{attribute 'linkalways'} 
{attribute 'no_explicit_call' := 'This FB is a CLASS and must be accessed using methods or properties'}
{attribute 'enable_dynamic_creation'}
FUNCTION_BLOCK DatatypeOperations
VAR
	operations : Stack;
END_VAR

METHOD PUBLIC AddMemoryCopyOperation
VAR_INPUT
	Source : I_Datatype;
	Destination : I_Datatype;
END_VAR
VAR
	operation : I_DatatypeOperation;
END_VAR
operation := CreateMemoryCopyOperation(Source,Destination);
operations.Push(operation);
END_METHOD

METHOD PUBLIC AddSafeMemoryCopyOperation
VAR_INPUT
	Source : I_Datatype;
	Destination : I_Datatype;
END_VAR
VAR
	operation : I_DatatypeOperation;
END_VAR
operation := CreateSafeMemoryCopyOperation(Source,Destination);
operations.Push(operation);
END_METHOD

METHOD PUBLIC AddWriteBitToBoolOperation
VAR_INPUT
	Source : I_BitDatatype;
	Destination : Reference to _BOOL;
END_VAR
VAR
	operation : I_DatatypeOperation;
END_VAR
operation := CreateWriteBitToBoolOperation(Source,Destination);
operations.Push(operation);
END_METHOD

METHOD PUBLIC AddWriteBoolToBitOperation
VAR_INPUT
	Source : REFERENCE TO _BOOL;
	Destination : I_BitDatatype;
END_VAR
VAR
	operation : I_DatatypeOperation;
END_VAR
operation := CreateWriteBoolToBitOperation(Source,Destination);
operations.Push(operation);
END_METHOD

METHOD PUBLIC Clear
VAR
	operation : I_DatatypeOperation;
END_VAR
WHILE operations.TryPop(operation) DO
	operation.Dispose();
END_WHILE
END_METHOD

METHOD PRIVATE CreateMemoryCopyOperation : I_DatatypeOperation
VAR_INPUT
	OperationSource : I_Datatype;
	OperationDestination : I_Datatype;
END_VAR
VAR
	pOperation : POINTER TO MemCopyOperation;
END_VAR
pOperation := __NEW(MemCopyOperation(Source := OperationSource, Destination := OperationDestination));
CreateMemoryCopyOperation := pOperation^;
END_METHOD

METHOD PRIVATE CreateSafeMemoryCopyOperation : I_DatatypeOperation
VAR_INPUT
	OperationSource : I_Datatype;
	OperationDestination : I_Datatype;
END_VAR
VAR
	pOperation : POINTER TO SafeMemCopyOperation;
END_VAR
pOperation := __NEW(SafeMemCopyOperation(Source := OperationSource, Destination := OperationDestination));
CreateSafeMemoryCopyOperation := pOperation^;
END_METHOD

METHOD PRIVATE CreateWriteBitToBoolOperation : I_DatatypeOperation
VAR_INPUT
	OperationSource : I_BitDatatype;
	OperationDestination : REFERENCE TO _BOOL;
END_VAR
VAR
	pOperation : POINTER TO WriteBitToBoolOperation;
END_VAR
pOperation := __NEW(WriteBitToBoolOperation(Source := OperationSource, Destination := OperationDestination));
CreateWriteBitToBoolOperation := pOperation^;
END_METHOD

METHOD PRIVATE CreateWriteBoolToBitOperation : I_DatatypeOperation
VAR_INPUT
	OperationSource : REFERENCE TO _BOOL;
	OperationDestination : I_BitDatatype;
END_VAR
VAR
	pOperation : POINTER TO WriteBoolToBitOperation;
END_VAR
pOperation := __NEW(WriteBoolToBitOperation(Source := OperationSource, Destination := OperationDestination));
CreateWriteBoolToBitOperation := pOperation^;
END_METHOD

METHOD PUBLIC Execute
VAR
	enumerator : I_ForwardEnumerator;
	operation : I_DatatypeOperation;
END_VAR
enumerator := operations.GetEnumerator();

WHILE enumerator.MoveNext() DO
	IF enumerator.TryGet(operation) THEN
		operation.Execute();
	END_IF
END_WHILE

enumerator.Dispose();
END_METHOD

METHOD FB_exit : BOOL
VAR_INPUT
	bInCopyCode : BOOL; // if TRUE, the exit method is called for exiting an instance that is copied afterwards (online change).
END_VAR
IF bInCopyCode THEN
	RETURN;
END_IF

operations.Clear();
END_METHOD

END_FUNCTION_BLOCK

(* stored: Version 1.1.0.1, ProductVersion 3.1.4024.12
   POU DatatypeOperations: Id {708b0684-560f-40e9-9f5c-eacc1f244428}, SpecialFunc None
   Folder Destructor: Id {e9d473f4-534f-48be-9ad9-8065a552fc27}
   Folder Private: Id {0618b737-9985-499e-9c25-c68bcb08b915}
   Method AddMemoryCopyOperation: Id {0b56884a-04bf-4df6-8151-73d98e4185b0}
   Method AddSafeMemoryCopyOperation: Id {33d58660-017d-46db-9c10-803ea54aae4e}
   Method AddWriteBitToBoolOperation: Id {b1df01cf-5dd7-413c-8414-ab9aae948c26}
   Method AddWriteBoolToBitOperation: Id {d4be1b58-d006-4f02-bc1f-dce058564e69}
   Method Clear: Id {c1a776d8-6574-44ae-ae04-07581ae56e57}
   Method CreateMemoryCopyOperation: Id {3ed42d4c-c19e-4091-a24b-e689760c3035}
   Method CreateSafeMemoryCopyOperation: Id {5e3b25fa-db01-4f2c-8df3-dac5b2a717de}
   Method CreateWriteBitToBoolOperation: Id {59f957cb-1c50-4fd8-b3e4-c6e1e7d519cf}
   Method CreateWriteBoolToBitOperation: Id {90e95abd-d6fb-4f00-b918-4d1da5d6e592}
   Method Execute: Id {0d36df40-f191-46a1-84c9-8d13d60c0338}
   Method FB_exit: Id {350f7d84-6ecb-4517-8681-368ca2861a92} *)
